PROGRAM MAIN
VAR
	{attribute 'TcHmiSystemEng.Parameter.Name' 				:= 'Machine'}
	{attribute 'TcHmiSystemEng.Parameter.TreeViewImage'	 	:= 'Portal/normal.svg'}	
	fbMachine					: FB_MachineUnit;
	
	_isInit      				: BOOL;
END_VAR

END_PROGRAM

(* stored: Version 1.1.0.1
   POU MAIN: Id {6897fa1c-d9fc-4690-9cab-da7b27af73be}, SpecialFunc None *)
